% RSLogix 500 project I2P Hands-On 4 - Caylen Johnson.RSS, saved by version 10.00.00.00 %
PROJECT "UNTITLED"    % processor: Bul.1763 MicroLogix 1100 Series B %

PROGRAM FILES
  LAD 2   14 rungs

DATA FILES
  O0 OUTPUT  4 elements
  I1 INPUT  6 elements
  S2 STATUS  66 elements
  B3 BINARY  1 elements
  T4 TIMER  1 elements
  C5 COUNTER  1 elements
  R6 CONTROL  1 elements
  N7 INTEGER  1 elements
  F8 FLOAT  1 elements

LADDER 2
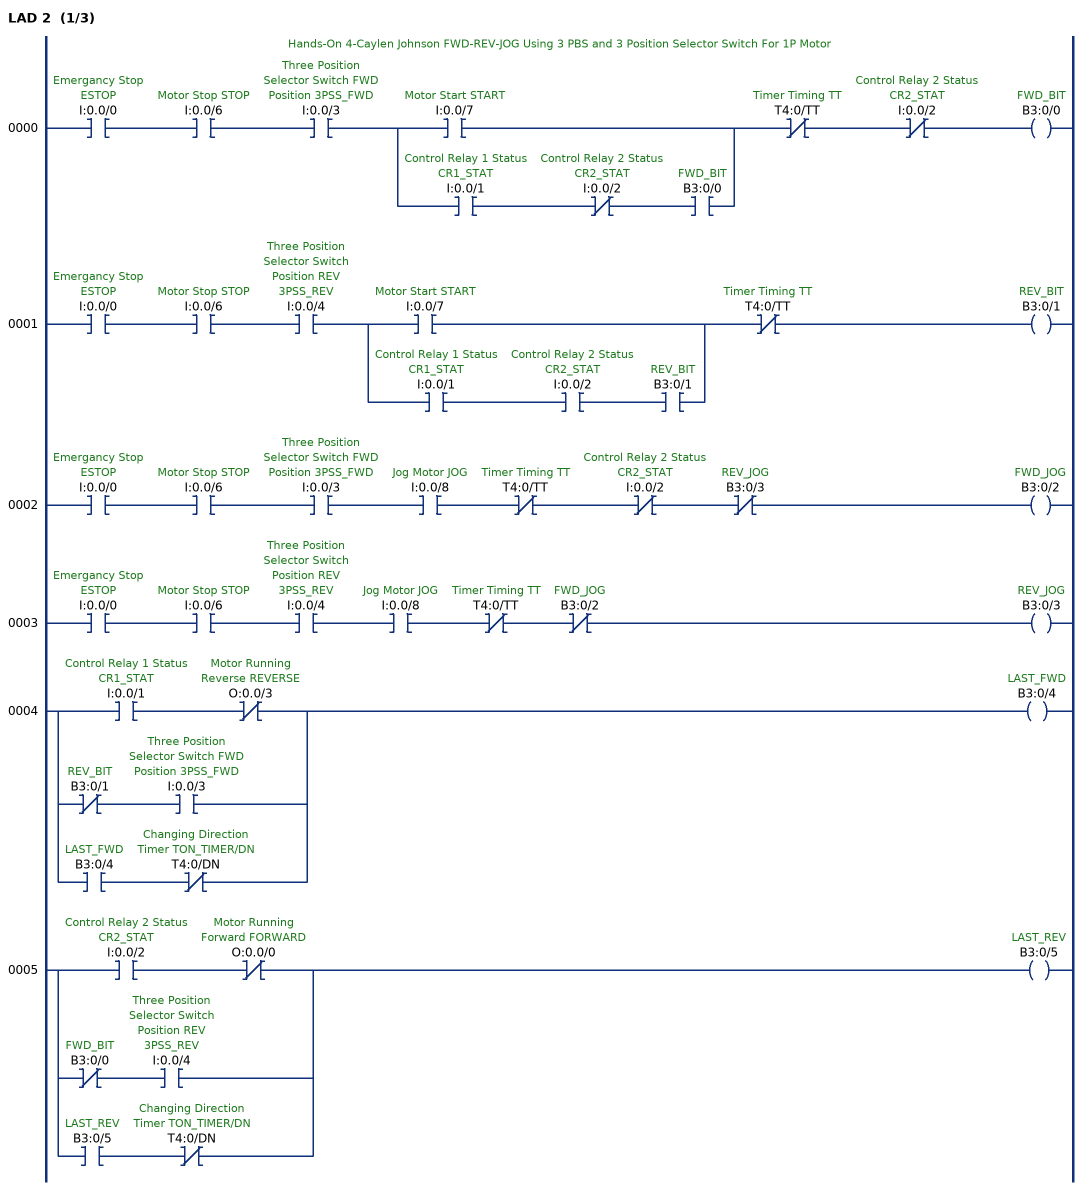
% Rung: 0 %
% Hands-On 4-Caylen Johnson FWD-REV-JOG Using 3 PBS and 3 Position Selector Switch For 1P Motor %
SOR XIC I:0.0/0 XIC I:0.0/6 XIC I:0.0/3 BST XIC I:0.0/7 NXB XIC I:0.0/1 XIO I:0.0/2 XIC B3:0/0 BND XIO T4:0/TT XIO I:0.0/2 OTE B3:0/0 EOR
%   I:0.0/0  ESTOP  "Emergancy Stop" %
%   I:0.0/6  STOP  "Motor Stop" %
%   I:0.0/3  3PSS_FWD  "Three Position Selector Switch FWD Position" %
%   I:0.0/7  START  "Motor Start" %
%   I:0.0/1  CR1_STAT  "Control Relay 1 Status" %
%   I:0.0/2  CR2_STAT  "Control Relay 2 Status" %
%   B3:0/0  FWD_BIT %
%   T4:0/TT  TT  "Timer Timing" %
% Rung: 1 %
SOR XIC I:0.0/0 XIC I:0.0/6 XIC I:0.0/4 BST XIC I:0.0/7 NXB XIC I:0.0/1 XIC I:0.0/2 XIC B3:0/1 BND XIO T4:0/TT OTE B3:0/1 EOR
%   I:0.0/0  ESTOP  "Emergancy Stop" %
%   I:0.0/6  STOP  "Motor Stop" %
%   I:0.0/4  3PSS_REV  "Three Position Selector Switch Position REV" %
%   I:0.0/7  START  "Motor Start" %
%   I:0.0/1  CR1_STAT  "Control Relay 1 Status" %
%   I:0.0/2  CR2_STAT  "Control Relay 2 Status" %
%   B3:0/1  REV_BIT %
%   T4:0/TT  TT  "Timer Timing" %
% Rung: 2 %
SOR XIC I:0.0/0 XIC I:0.0/6 XIC I:0.0/3 XIC I:0.0/8 XIO T4:0/TT XIO I:0.0/2 XIO B3:0/3 OTE B3:0/2 EOR
%   I:0.0/0  ESTOP  "Emergancy Stop" %
%   I:0.0/6  STOP  "Motor Stop" %
%   I:0.0/3  3PSS_FWD  "Three Position Selector Switch FWD Position" %
%   I:0.0/8  JOG  "Jog Motor" %
%   T4:0/TT  TT  "Timer Timing" %
%   I:0.0/2  CR2_STAT  "Control Relay 2 Status" %
%   B3:0/3  REV_JOG %
%   B3:0/2  FWD_JOG %
% Rung: 3 %
SOR XIC I:0.0/0 XIC I:0.0/6 XIC I:0.0/4 XIC I:0.0/8 XIO T4:0/TT XIO B3:0/2 OTE B3:0/3 EOR
%   I:0.0/0  ESTOP  "Emergancy Stop" %
%   I:0.0/6  STOP  "Motor Stop" %
%   I:0.0/4  3PSS_REV  "Three Position Selector Switch Position REV" %
%   I:0.0/8  JOG  "Jog Motor" %
%   T4:0/TT  TT  "Timer Timing" %
%   B3:0/2  FWD_JOG %
%   B3:0/3  REV_JOG %
% Rung: 4 %
SOR BST XIC I:0.0/1 XIO O:0.0/3 NXB BST XIO B3:0/1 XIC I:0.0/3 NXB XIC B3:0/4 XIO T4:0/DN BND BND OTE B3:0/4 EOR
%   I:0.0/1  CR1_STAT  "Control Relay 1 Status" %
%   O:0.0/3  REVERSE  "Motor Running Reverse" %
%   B3:0/1  REV_BIT %
%   I:0.0/3  3PSS_FWD  "Three Position Selector Switch FWD Position" %
%   B3:0/4  LAST_FWD %
%   T4:0  TON_TIMER  "Changing Direction Timer" %
% Rung: 5 %
SOR BST XIC I:0.0/2 XIO O:0.0/0 NXB BST XIO B3:0/0 XIC I:0.0/4 NXB XIC B3:0/5 XIO T4:0/DN BND BND OTE B3:0/5 EOR
%   I:0.0/2  CR2_STAT  "Control Relay 2 Status" %
%   O:0.0/0  FORWARD  "Motor Running Forward" %
%   B3:0/0  FWD_BIT %
%   I:0.0/4  3PSS_REV  "Three Position Selector Switch Position REV" %
%   B3:0/5  LAST_REV %
%   T4:0  TON_TIMER  "Changing Direction Timer" %

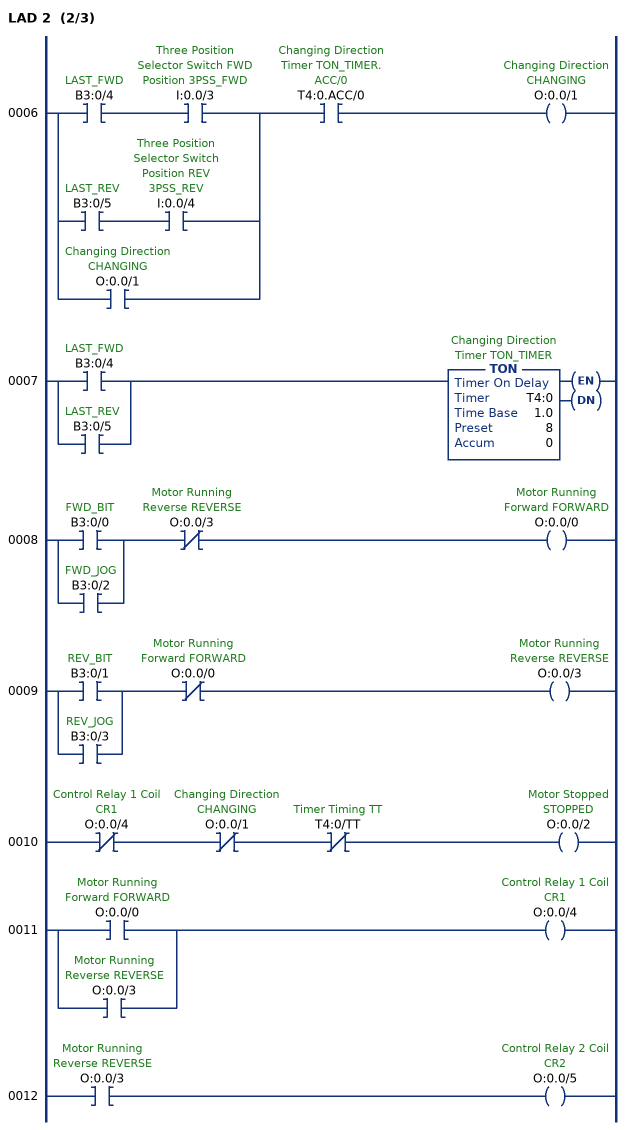
% Rung: 6 %
SOR BST XIC B3:0/4 XIC I:0.0/3 NXB BST XIC B3:0/5 XIC I:0.0/4 NXB XIC O:0.0/1 BND BND XIC T4:0.ACC/0 OTE O:0.0/1 EOR
%   B3:0/4  LAST_FWD %
%   I:0.0/3  3PSS_FWD  "Three Position Selector Switch FWD Position" %
%   B3:0/5  LAST_REV %
%   I:0.0/4  3PSS_REV  "Three Position Selector Switch Position REV" %
%   O:0.0/1  CHANGING  "Changing Direction" %
%   T4:0  TON_TIMER  "Changing Direction Timer" %
% Rung: 7 %
SOR BST XIC B3:0/4 NXB XIC B3:0/5 BND TON T4:0 1.0 8 0 EOR
%   B3:0/4  LAST_FWD %
%   B3:0/5  LAST_REV %
%   T4:0  TON_TIMER  "Changing Direction Timer" %
% Rung: 8 %
SOR BST XIC B3:0/0 NXB XIC B3:0/2 BND XIO O:0.0/3 OTE O:0.0/0 EOR
%   B3:0/0  FWD_BIT %
%   B3:0/2  FWD_JOG %
%   O:0.0/3  REVERSE  "Motor Running Reverse" %
%   O:0.0/0  FORWARD  "Motor Running Forward" %
% Rung: 9 %
SOR BST XIC B3:0/1 NXB XIC B3:0/3 BND XIO O:0.0/0 OTE O:0.0/3 EOR
%   B3:0/1  REV_BIT %
%   B3:0/3  REV_JOG %
%   O:0.0/0  FORWARD  "Motor Running Forward" %
%   O:0.0/3  REVERSE  "Motor Running Reverse" %
% Rung: 10 %
SOR XIO O:0.0/4 XIO O:0.0/1 XIO T4:0/TT OTE O:0.0/2 EOR
%   O:0.0/4  CR1  "Control Relay 1 Coil" %
%   O:0.0/1  CHANGING  "Changing Direction" %
%   T4:0/TT  TT  "Timer Timing" %
%   O:0.0/2  STOPPED  "Motor Stopped" %
% Rung: 11 %
SOR BST XIC O:0.0/0 NXB XIC O:0.0/3 BND OTE O:0.0/4 EOR
%   O:0.0/0  FORWARD  "Motor Running Forward" %
%   O:0.0/3  REVERSE  "Motor Running Reverse" %
%   O:0.0/4  CR1  "Control Relay 1 Coil" %
% Rung: 12 %
SOR XIC O:0.0/3 OTE O:0.0/5 EOR
%   O:0.0/3  REVERSE  "Motor Running Reverse" %
%   O:0.0/5  CR2  "Control Relay 2 Coil" %

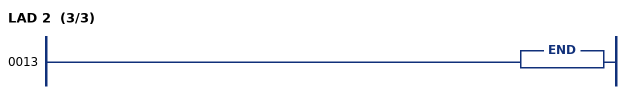
% Rung: 13 %
SOR END EOR

DATA TABLE (non-zero values as saved)
DATA B3
% B3:0 % 0X0010
DATA T4
% .PRE .ACC %
% T4:0 % 8 0
